Fanuc KAREL source: picking_point_parser.kl

PROGRAM picking_point_parser
%NOLOCKGROUP
%NOBUSYLAMP

TYPE
    picking_point = STRUCTURE
        picker_position: XYZWPR
    ENDSTRUCTURE

VAR
 	 test_json : STRING[40]
 	 res : picking_point

ROUTINE parsePickingPoint(original_text: STRING; text_index: INTEGER) : picking_point
----------------------------------------------------
-- Creation date: 2020.04.15
-- Created by:
----------------------------------------------------
-- Function:
----------------------------------------------------
-- Arguments:
----------------------------------------------------
-- Return value:
----------------------------------------------------
-- Last modified: 2020.04.15
-- Last modified by:
----------------------------------------------------

	VAR
	    x : REAL
	    y : REAL
	    z : REAL
	    w : REAL
	    p : REAL
	    r : REAL
	    c : STRING[1]
	    c_1 : STRING[1]
	    string_value : STRING[20]
	    key_pointer : INTEGER
	    searching : BOOLEAN
	    candidate : STRING[3]
	    loop1 : BOOLEAN
	    reading : BOOLEAN
	    v : REAL
	    ret_val : picking_point
	BEGIN
	    searching = TRUE
	    key_pointer = 0
	    candidate = ''
	    loop1 = TRUE
	    reading = FALSE
	    string_value = ''
	    -- prints for testing
	    WRITE(original_text, text_index)
	    WHILE loop1 = TRUE DO
	    	 c = SUB_STR(original_text, text_index, 1)
	        text_index = text_index + 1
	        IF searching = TRUE THEN
	            IF (((key_pointer = 0) OR (key_pointer = 2)) AND (c = '"')) OR ((key_pointer = 1) AND ((c = 'x') OR (c = 'y') OR (c = 'z') OR (c = 'w') OR (c = 'p') OR (c = 'r'))) THEN
	                candidate = candidate + c -- string sum
	                key_pointer = key_pointer + 1
	            ELSE
	                candidate = ''
	                key_pointer = 0
	            ENDIF
	            IF key_pointer = 3 THEN
	                searching = FALSE
	                key_pointer = 0
	                c_1 = SUB_STR(candidate, 1, 1)
	            ENDIF
	        ELSE -- we found our candidate
	            IF (reading = TRUE) AND (c <> ' ') AND (c <> ',') AND (c <> '}') THEN
	                string_value = string_value + c -- string sum
	            ENDIF
	            IF c = ':' THEN
	                reading = TRUE
	            ENDIF
	            IF (c = ',') OR (c = '}') THEN
	                searching = TRUE
	                reading = FALSE
	                v = 0
	                CNV_STR_REAL(string_value, v) -- v = real(string_value)
	                IF  c_1 = 'x' THEN
	                    x = v
	                ENDIF
	                IF  c_1 = 'y' THEN
	                    y = v
	                ENDIF
	                IF  c_1 = 'z' THEN
	                    z = v
	                ENDIF
	                IF c_1 = 'w' THEN
	                    w = v
	                ENDIF
	                IF  c_1 = 'p' THEN
	                    p = v
	                ENDIF
	                IF  c_1 = 'r' THEN
	                    r = v
	                ENDIF
	                candidate = ''
	            ENDIF
	            IF c = '}' THEN
	                ret_val.picker_position.x = x
	                ret_val.picker_position.y = y
	                ret_val.picker_position.z = z
	                ret_val.picker_position.w = w
	                ret_val.picker_position.p = p
	                ret_val.picker_position.r = r
	                loop1 = FALSE
	            ENDIF
	        ENDIF
	    ENDWHILE
	    RETURN (ret_val)
	END parsePickingPoint

BEGIN
    test_json = '{"x":0, "y":0, "z":0, "w":0, "p":0, "r":0}'
    res =  parsePickingPoint(test_json, 1)
    WRITE(res)
END picking_point_parser
